// TIA Portal project "Final Project" (V15.1)

(* hardware
DEVICE "S7-1200 station_1"  S7-1200 Station
   slot 0: "Rack_0"  S7-1200 Rack  Rack  V1.0
   slot 1: "PLC_1"  CPU 1214C AC/DC/Rly  6ES7 214-1BG31-0XB0  V3.0
   slot 3: "AQ 1x12BIT_1"  AQ1 signal board  6ES7 232-4HA30-0XB0  V1.0
*)

// ===== PLC "PLC_1"  CPU 1214C AC/DC/Rly =====

VAR_GLOBAL   // PLC tag table "Default tag table"
   "b_sto" AT %I0.1 : Bool;
   "b_sta" AT %I0.2 : Bool;
   "b_slo" AT %I0.3 : Bool;
   "b_fas" AT %I0.4 : Bool;
   "b_eme" AT %I0.0 : Bool;
   "b_a" AT %I0.6 : Bool;
   "c_sta" AT %M0.1 : Bool;
   "L_y" AT %Q0.1 : Bool;
   "L_g" AT %Q0.0 : Bool;
   "L_r" AT %Q0.2 : Bool;
   "n" AT %M0.3 : Bool;
   "h_l" AT %M0.5 : Bool;
   "h_s" AT %M0.6 : Bool;
   "P_se" AT %Q0.7 : Bool;
   "P_sc" AT %Q0.6 : Bool;
   "P_le" AT %Q1.1 : Bool;
   "P_lc" AT %Q1.0 : Bool;
   "A" AT %M2.2 : Bool;
   "B" AT %M2.3 : Bool;
   "C" AT %M2.4 : Bool;
   "D" AT %M2.5 : Bool;
   "b_m" AT %I0.5 : Bool;
   "E" AT %M1.7 : Bool;
   "F" AT %M1.0 : Bool;
   "G" AT %M1.1 : Bool;
   "H" AT %M1.2 : Bool;
   "I" AT %M1.3 : Bool;
   "s1" AT %Q0.3 : Bool;
   "s2" AT %Q0.4 : Bool;
   "s3" AT %Q0.5 : Bool;
   "A_lamp" AT %M2.6 : Bool;
   "B_lamp" AT %M2.7 : Bool;
   "h_la" AT %IW66 : Int;
   "h_sa" AT %IW64 : Int;
END_VAR

// folder: System blocks/Program resources

DATA_BLOCK "T_s2"   // DB1
{ S7_Optimized_Access := 'TRUE' }
AUTHOR : Simatic
FAMILY : IEC
NAME : IEC_TMR
VERSION : 1.0
// stored: InstanceOfName IEC_TIMER
"IEC_TIMER"
BEGIN
END_DATA_BLOCK

DATA_BLOCK "T_y1"   // DB2
{ S7_Optimized_Access := 'TRUE' }
AUTHOR : Simatic
FAMILY : IEC
NAME : IEC_TMR
VERSION : 1.0
// stored: InstanceOfName IEC_TIMER
"IEC_TIMER"
BEGIN
END_DATA_BLOCK

DATA_BLOCK "T_y2"   // DB3
{ S7_Optimized_Access := 'TRUE' }
AUTHOR : Simatic
FAMILY : IEC
NAME : IEC_TMR
VERSION : 1.0
// stored: InstanceOfName IEC_TIMER
"IEC_TIMER"
BEGIN
END_DATA_BLOCK

DATA_BLOCK "T_g1"   // DB4
{ S7_Optimized_Access := 'TRUE' }
AUTHOR : Simatic
FAMILY : IEC
NAME : IEC_TMR
VERSION : 1.0
// stored: InstanceOfName IEC_TIMER
"IEC_TIMER"
BEGIN
END_DATA_BLOCK

DATA_BLOCK "T_g2"   // DB5
{ S7_Optimized_Access := 'TRUE' }
AUTHOR : Simatic
FAMILY : IEC
NAME : IEC_TMR
VERSION : 1.0
// stored: InstanceOfName IEC_TIMER
"IEC_TIMER"
BEGIN
END_DATA_BLOCK

DATA_BLOCK "T_r1"   // DB6
{ S7_Optimized_Access := 'TRUE' }
AUTHOR : Simatic
FAMILY : IEC
NAME : IEC_TMR
VERSION : 1.0
// stored: InstanceOfName IEC_TIMER
"IEC_TIMER"
BEGIN
END_DATA_BLOCK

DATA_BLOCK "T_r2"   // DB7
{ S7_Optimized_Access := 'TRUE' }
AUTHOR : Simatic
FAMILY : IEC
NAME : IEC_TMR
VERSION : 1.0
// stored: InstanceOfName IEC_TIMER
"IEC_TIMER"
BEGIN
END_DATA_BLOCK

DATA_BLOCK "T_s"   // DB8
{ S7_Optimized_Access := 'TRUE' }
AUTHOR : Simatic
FAMILY : IEC
NAME : IEC_TMR
VERSION : 1.0
// stored: InstanceOfName IEC_TIMER
"IEC_TIMER"
BEGIN
END_DATA_BLOCK

DATA_BLOCK "T_l"   // DB9
{ S7_Optimized_Access := 'TRUE' }
AUTHOR : Simatic
FAMILY : IEC
NAME : IEC_TMR
VERSION : 1.0
// stored: InstanceOfName IEC_TIMER
"IEC_TIMER"
BEGIN
END_DATA_BLOCK

DATA_BLOCK "T_c"   // DB10
{ S7_Optimized_Access := 'TRUE' }
AUTHOR : Simatic
FAMILY : IEC
NAME : IEC_TMR
VERSION : 1.0
// stored: InstanceOfName IEC_TIMER
"IEC_TIMER"
BEGIN
END_DATA_BLOCK

DATA_BLOCK "T_l2"   // DB11
{ S7_Optimized_Access := 'TRUE' }
AUTHOR : Simatic
FAMILY : IEC
NAME : IEC_TMR
VERSION : 1.0
// stored: InstanceOfName IEC_TIMER
"IEC_TIMER"
BEGIN
END_DATA_BLOCK

// folder: (top level)

ORGANIZATION_BLOCK "Main"   // OB1, LAD, ProgramCycle
TITLE = "Main Program Sweep (Cycle)"
{ S7_Optimized_Access := 'TRUE' }
VERSION : 0.1
   VAR_TEMP   // added for the SCL form of the ladder/FBD networks
      _w1 : Bool;
   END_VAR
BEGIN

REGION Network 1: Conveyor belt
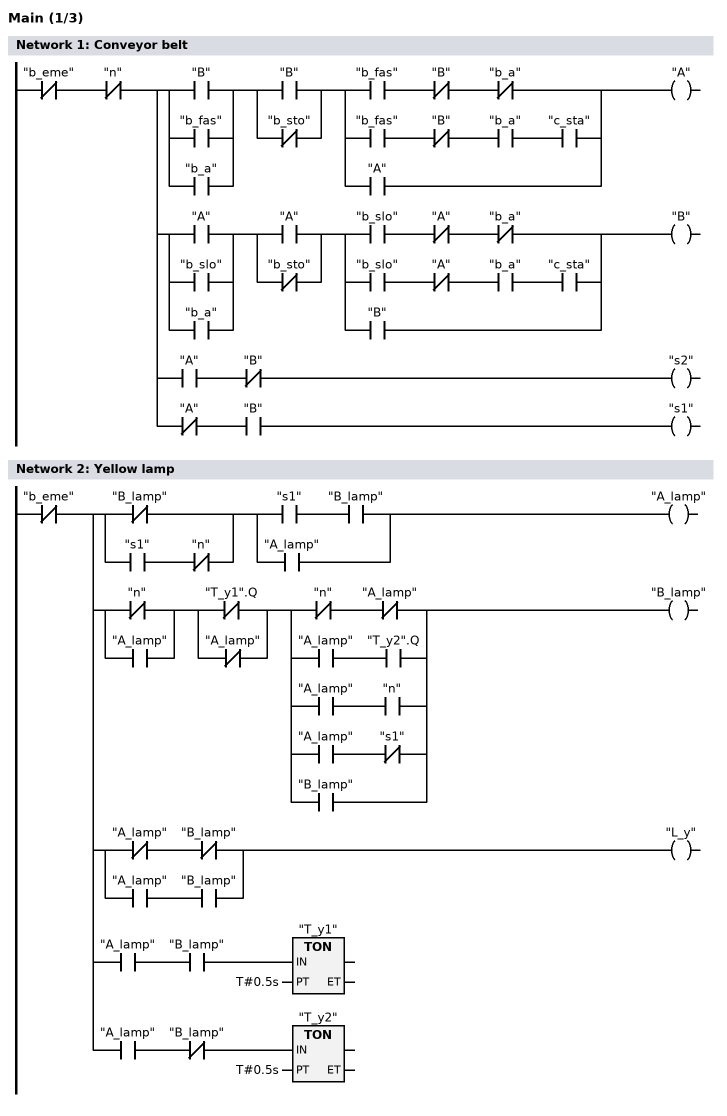
   RUNG wire#powerrail
      I_Contact( "b_eme" )
      I_Contact( "n" )
      wire#w1
      Contact( "B" )
      wire#w2
      Contact( "B" )
      wire#w3
      Contact( "b_fas" )
      I_Contact( "B" )
      I_Contact( "b_a" )
      wire#w4
      Coil( "A" )
   END_RUNG
   RUNG wire#w1
      Contact( "b_fas" )
   END_RUNG wire#w2
   RUNG wire#w1
      Contact( "b_a" )
   END_RUNG wire#w2
   RUNG wire#w2
      I_Contact( "b_sto" )
   END_RUNG wire#w3
   RUNG wire#w3
      Contact( "b_fas" )
      I_Contact( "B" )
      Contact( "b_a" )
      Contact( "c_sta" )
   END_RUNG wire#w4
   RUNG wire#w3
      Contact( "A" )
   END_RUNG wire#w4
   RUNG wire#w1
      Contact( "A" )
      wire#w5
      Contact( "A" )
      wire#w6
      Contact( "b_slo" )
      I_Contact( "A" )
      I_Contact( "b_a" )
      wire#w7
      Coil( "B" )
   END_RUNG
   RUNG wire#w1
      Contact( "b_slo" )
   END_RUNG wire#w5
   RUNG wire#w1
      Contact( "b_a" )
   END_RUNG wire#w5
   RUNG wire#w5
      I_Contact( "b_sto" )
   END_RUNG wire#w6
   RUNG wire#w6
      Contact( "b_slo" )
      I_Contact( "A" )
      Contact( "b_a" )
      Contact( "c_sta" )
   END_RUNG wire#w7
   RUNG wire#w6
      Contact( "B" )
   END_RUNG wire#w7
   RUNG wire#w1
      Contact( "A" )
      I_Contact( "B" )
      Coil( "s2" )
   END_RUNG
   RUNG wire#w1
      I_Contact( "A" )
      Contact( "B" )
      Coil( "s1" )
   END_RUNG
   // the same network as SCL:
   #_w1 := NOT "b_eme" AND NOT "n";
   "A" := #_w1 AND ("B" OR "b_fas" OR "b_a") AND ("B" OR NOT "b_sto") AND (("b_fas" AND NOT "B" AND NOT "b_a") OR ("b_fas" AND NOT "B" AND "b_a" AND "c_sta") OR "A");
   "B" := #_w1 AND ("A" OR "b_slo" OR "b_a") AND ("A" OR NOT "b_sto") AND (("b_slo" AND NOT "A" AND NOT "b_a") OR ("b_slo" AND NOT "A" AND "b_a" AND "c_sta") OR "B");
   "s2" := #_w1 AND "A" AND NOT "B";
   "s1" := #_w1 AND NOT "A" AND "B";
END_REGION

REGION Network 2: Yellow lamp
   "A_lamp" := NOT "b_eme" AND (NOT "B_lamp" OR ("s1" AND NOT "n")) AND (("s1" AND "B_lamp") OR "A_lamp");
   "B_lamp" := NOT "b_eme" AND (NOT "n" OR "A_lamp") AND (NOT "T_y1".Q OR NOT "A_lamp") AND ((NOT "n" AND NOT "A_lamp") OR ("A_lamp" AND "T_y2".Q) OR ("A_lamp" AND "n") OR ("A_lamp" AND NOT "s1") OR "B_lamp");
   "L_y" := NOT "b_eme" AND ((NOT "A_lamp" AND NOT "B_lamp") OR ("A_lamp" AND "B_lamp"));
   "T_y1".TON(IN := NOT "b_eme" AND "A_lamp" AND "B_lamp", PT := T#0.5s);
   "T_y2".TON(IN := NOT "b_eme" AND "A_lamp" AND NOT "B_lamp", PT := T#0.5s);
END_REGION

REGION Network 3: Green lamp
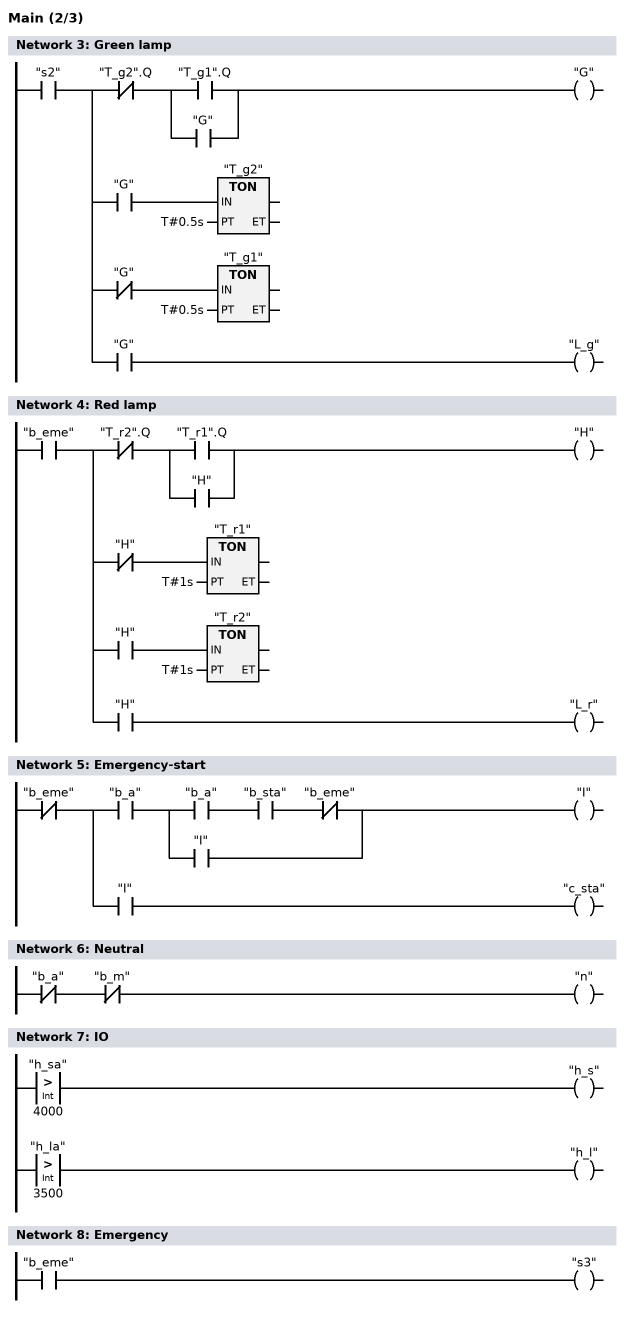
   "G" := "s2" AND NOT "T_g2".Q AND ("T_g1".Q OR "G");
   "T_g2".TON(IN := "s2" AND "G", PT := T#0.5s);
   "T_g1".TON(IN := "s2" AND NOT "G", PT := T#0.5s);
   "L_g" := "s2" AND "G";
END_REGION

REGION Network 4: Red lamp
   "H" := "b_eme" AND NOT "T_r2".Q AND ("T_r1".Q OR "H");
   "T_r1".TON(IN := "b_eme" AND NOT "H", PT := T#1s);
   "T_r2".TON(IN := "b_eme" AND "H", PT := T#1s);
   "L_r" := "b_eme" AND "H";
END_REGION

REGION Network 5: Emergency-start
   RUNG wire#powerrail
      I_Contact( "b_eme" )
      wire#w1
      Contact( "b_a" )
      wire#w2
      Contact( "b_a" )
      Contact( "b_sta" )
      I_Contact( "b_eme" )
      wire#w3
      Coil( "I" )
   END_RUNG
   RUNG wire#w2
      Contact( "I" )
   END_RUNG wire#w3
   RUNG wire#w1
      Contact( "I" )
      Coil( "c_sta" )
   END_RUNG
   // the same network as SCL:
   "I" := NOT "b_eme" AND "b_a" AND (("b_a" AND "b_sta" AND NOT "b_eme") OR "I");
   "c_sta" := NOT "b_eme" AND "I";
END_REGION

REGION Network 6: Neutral
   RUNG wire#powerrail
      I_Contact( "b_a" )
      I_Contact( "b_m" )
      Coil( "n" )
   END_RUNG
   // the same network as SCL:
   "n" := NOT "b_a" AND NOT "b_m";
END_REGION

REGION Network 7: IO
   RUNG wire#powerrail
      { S7_Templates := "SrcType := Int" } GT_Contact(in1 := "h_sa", in2 := 4000)
      Coil( "h_s" )
   END_RUNG
   RUNG wire#powerrail
      { S7_Templates := "SrcType := Int" } GT_Contact(in1 := "h_la", in2 := 3500)
      Coil( "h_l" )
   END_RUNG
   // the same network as SCL:
   "h_s" := "h_sa" > 4000;
   "h_l" := "h_la" > 3500;
END_REGION

REGION Network 8: Emergency
   RUNG wire#powerrail
      Contact( "b_eme" )
      Coil( "s3" )
   END_RUNG
   // the same network as SCL:
   "s3" := "b_eme";
END_REGION

REGION Network 9: Pistons ver 2
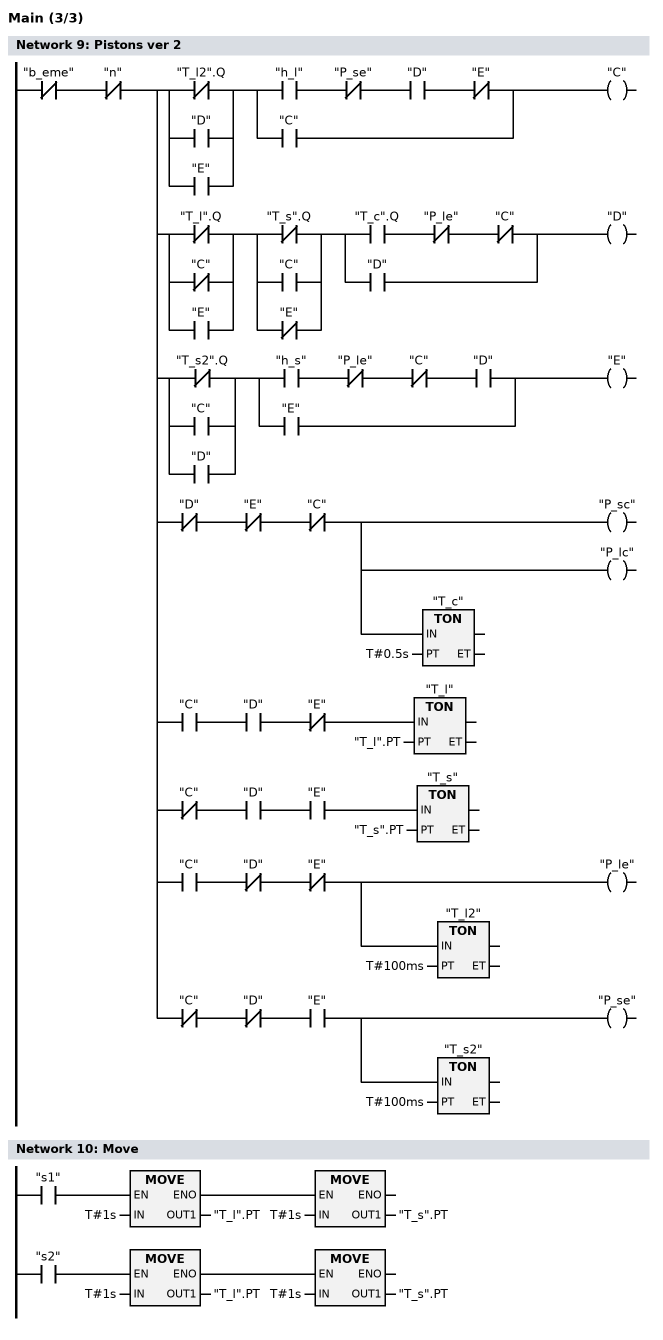
   #_w1 := NOT "b_eme" AND NOT "n";
   "C" := #_w1 AND (NOT "T_l2".Q OR "D" OR "E") AND (("h_l" AND NOT "P_se" AND "D" AND NOT "E") OR "C");
   "D" := #_w1 AND (NOT "T_l".Q OR NOT "C" OR "E") AND (NOT "T_s".Q OR "C" OR NOT "E") AND (("T_c".Q AND NOT "P_le" AND NOT "C") OR "D");
   "E" := #_w1 AND (NOT "T_s2".Q OR "C" OR "D") AND (("h_s" AND NOT "P_le" AND NOT "C" AND "D") OR "E");
   "P_sc" := #_w1 AND NOT "D" AND NOT "E" AND NOT "C";
   "P_lc" := "P_sc";
   "T_c".TON(IN := "P_sc", PT := T#0.5s);
   "T_l".TON(IN := #_w1 AND "C" AND "D" AND NOT "E", PT := "T_l".PT);
   "T_s".TON(IN := #_w1 AND NOT "C" AND "D" AND "E", PT := "T_s".PT);
   "P_le" := #_w1 AND "C" AND NOT "D" AND NOT "E";
   "T_l2".TON(IN := "P_le", PT := T#100ms);
   "P_se" := #_w1 AND NOT "C" AND NOT "D" AND "E";
   "T_s2".TON(IN := "P_se", PT := T#100ms);
END_REGION

REGION Network 10: Move
   RUNG wire#powerrail
      Contact( "s1" )
      { S7_GenerateENO := "TRUE" } Move(in := T#1s, out1 => "T_l".PT)
      { S7_GenerateENO := "TRUE" } Move(in := T#1s, out1 => "T_s".PT)
   END_RUNG
   RUNG wire#powerrail
      Contact( "s2" )
      { S7_GenerateENO := "TRUE" } Move(in := T#1s, out1 => "T_l".PT)
      { S7_GenerateENO := "TRUE" } Move(in := T#1s, out1 => "T_s".PT)
   END_RUNG
   // the same network as SCL:
   // ENO of a box is taken as its EN; it also drops when the box reports an error
   IF "s1" THEN
       "T_l".PT := T#1s;
       "T_s".PT := T#1s;
   END_IF;
   IF "s2" THEN
       "T_l".PT := T#1s;
       "T_s".PT := T#1s;
   END_IF;
END_REGION
END_ORGANIZATION_BLOCK